RoboDK station: paint_robot.rdk

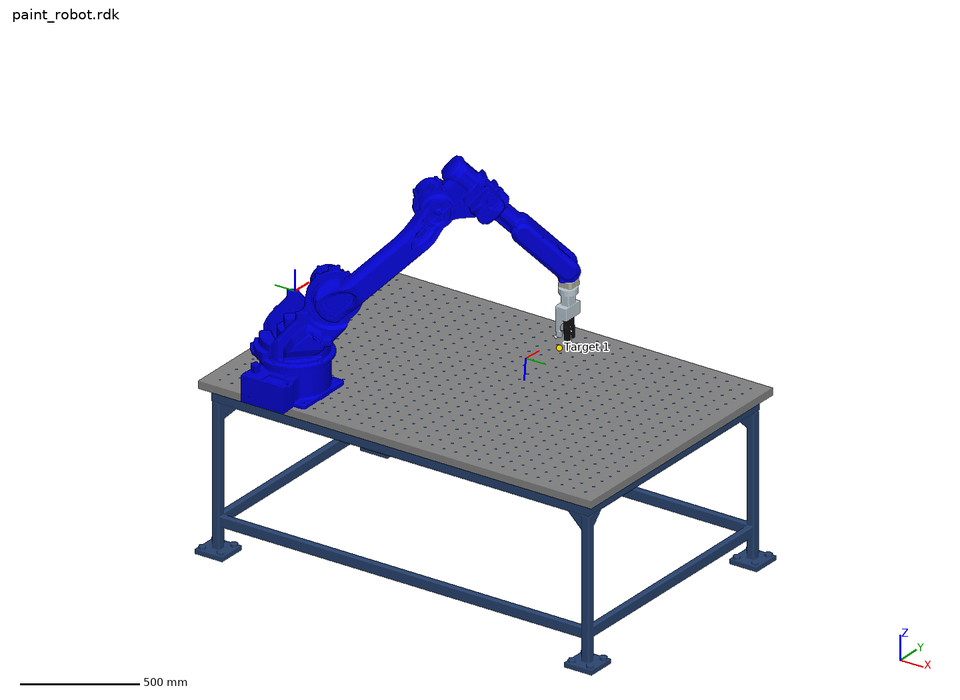
[picture v0: the station drawn from its stored meshes, robots at their saved joint values, targets as dots, program paths as lines]
Station paint_robot (saved by RoboDK 5.9.4). Poses are relative to the parent item; angles as X-Y-Z fixed-axis rotations.
  - frame Motoman HP6 Base at (2.87, -486.59, 450) mm, rotated rx 0 ry 0 rz 90.34 deg
    - robot Motoman HP6: 6 axes, payload 6 kg, reach 1378 mm, repeatability 0.08 mm, weight 130 kg
        modified DH rows (alpha deg, a mm, theta deg, d mm): 0, 0, 0, 450; -90, 150, -90, 0; 0, 570, 0, 0; -90, 155, 0, 640; 90, 0, 90, 0; -90, 0, 0, 95
        base shift (0, 0, -450) mm
        joint limits [-170, -90, -175, -180, -45, -360] to [170, 155, 250, 180, 225, 360]; home [0, 0, 0, 0, 0, 0]; saved at [-45.466, 50.692, 5.583, -1.431, 46.54, -134.308]
      - tool marker, TCP at (44.76, 5.33, 242.91) mm, size 100 x 89.2 x 281.5 mm
  - object table_draw at (0, 0, 0) mm, size 2020 x 1340 x 800 mm, geometry from Table-2000x1200x800mm.sld
  - frame Frame 2 at (685.28, 213.49, 50.15) mm, rotated rx -179.63 ry 3.79 rz 90.34 deg
    - target Target 1 (Cartesian target) at (108.07, 94.31, -36.38) mm, rotated rx 0.63 ry -5.51 rz -179.24 deg; joints [-43.036, 53.346, 5.286, -1.421, 49.532, -136.696] of Motoman HP6
  - Python program Prog1 (listed below)

--- Python program Prog1 ---
# draw_png_hp6_table_frame2.py
# Draw a PNG using Motoman HP6 in RoboDK (simulation).
# Station requirements:
#   Robot:       "Motoman HP6"
#   Tool:        "marker"
#   Draw frame:  "Frame 2"   -> XY plane of the paper
#   Base target: "DrawBase"  -> TCP at drawing height near center

from robolink import *   # RoboDK API
from robodk import *     # Pose tools
from robolink import TargetReachError

import cv2
import numpy as np
import os

# ---------------- CONFIG ----------------

IMAGE_PATH = r"vgtu.png"   # path to your PNG

ROBOT_NAME          = "Motoman HP6"
TOOL_NAME           = "marker"
DRAW_FRAME_NAME     = "Frame 2"
DRAW_BASE_TARGET    = "Target 1"

DRAW_AREA_MM = 150.0
MM_PER_PIXEL = 0.5     # scale of the drawing (mm per pixel)
POINT_STEP   = 4        # sample every Nth point of each contour

Z_DRAW  = 0.0           # drawing plane (relative to DrawBase)
Z_LIFT  = -50.0          # pen-up height above drawing plane (mm)

SPEED_DRAW   = 50.0     # mm/s when drawing
SPEED_TRAVEL = 200.0    # mm/s when travelling pen-up

# ----------------------------------------


def get_items(RDK: Robolink):
    """Get robot, tool, draw frame and base target from the station."""
    robot = RDK.Item(ROBOT_NAME, ITEM_TYPE_ROBOT)
    if not robot.Valid():
        raise Exception(f"Robot '{ROBOT_NAME}' not found in the station.")

    tool = RDK.Item(TOOL_NAME, ITEM_TYPE_TOOL)
    if not tool.Valid():
        raise Exception(f"Tool '{TOOL_NAME}' not found in the station.")

    draw_frame = RDK.Item(DRAW_FRAME_NAME, ITEM_TYPE_FRAME)
    if not draw_frame.Valid():
        raise Exception(f"Frame '{DRAW_FRAME_NAME}' (draw frame) not found.")

    base_target = RDK.Item(DRAW_BASE_TARGET, ITEM_TYPE_TARGET)
    if not base_target.Valid():
        raise Exception(
            f"Target '{DRAW_BASE_TARGET}' not found. "
            f"Teach it with the marker on the paper, near the center."
        )

    # Use our tool and draw frame for the robot
    robot.setPoseTool(tool)
    robot.setPoseFrame(draw_frame)

    return robot, draw_frame, base_target


def load_and_vectorize_image(image_path, draw_area_mm=DRAW_AREA_MM, point_step=4):
    """
    Load PNG, binarize it, find external contours and convert them
    to lists of XY points in mm, scaled to fit inside a square
    of size draw_area_mm x draw_area_mm and centered at (0,0).
    Returns: list of (N_i x 2) numpy arrays.
    """
    if not os.path.isfile(image_path):
        raise FileNotFoundError(f"Image not found: {image_path}")

    img = cv2.imread(image_path, cv2.IMREAD_GRAYSCALE)
    if img is None:
        raise Exception(f"Failed to read image: {image_path}")

    h, w = img.shape

    # Threshold: dark pixels become "ink"
    _, th = cv2.threshold(img, 200, 255, cv2.THRESH_BINARY_INV)

    contours, _ = cv2.findContours(th, cv2.RETR_EXTERNAL, cv2.CHAIN_APPROX_NONE)

    if not contours:
        raise Exception(
            "No drawing paths found in the image. "
            "Is the image mostly white/empty or too light?"
        )

    # --- collect all contour points in pixels to compute bounding box ---
    all_x = []
    all_y = []
    for cnt in contours:
        if len(cnt) < 5:
            continue
        xs = cnt[:, 0, 0]
        ys = cnt[:, 0, 1]
        all_x.append(xs)
        all_y.append(ys)

    all_x = np.concatenate(all_x).astype(np.float32)
    all_y = np.concatenate(all_y).astype(np.float32)

    xmin, xmax = all_x.min(), all_x.max()
    ymin, ymax = all_y.min(), all_y.max()

    cx = 0.5 * (xmin + xmax)
    cy = 0.5 * (ymin + ymax)

    span_x = xmax - xmin
    span_y = ymax - ymin
    span = max(span_x, span_y, 1e-6)   # avoid /0

    # scale so max dimension = draw_area_mm
    scale = float(draw_area_mm) / span

    paths_mm = []

    for cnt in contours:
        if len(cnt) < 5:
            continue

        pts = []
        for i in range(0, len(cnt), point_step):
            x_px = float(cnt[i][0][0])
            y_px = float(cnt[i][0][1])

            # center and scale; flip Y so "up" in image is +Y in frame
            x_mm = (x_px - cx) * scale
            y_mm = (y_px - cy) * scale

            pts.append([x_mm, y_mm])

        if len(pts) > 1:
            paths_mm.append(np.array(pts, dtype=float))

    if not paths_mm:
        raise Exception("Contours found, but no paths after processing.")

    # Optional: debug print to see range
    all_mm = np.vstack(paths_mm)
    print(
        f"[DEBUG] Drawing bounds in mm: "
        f"X [{all_mm[:,0].min():.1f}, {all_mm[:,0].max():.1f}], "
        f"Y [{all_mm[:,1].min():.1f}, {all_mm[:,1].max():.1f}]"
    )

    return paths_mm

# --------- motion helpers ---------

def move_pen_up(robot, base_pose, x_mm, y_mm, z_lift=Z_LIFT, speed=SPEED_TRAVEL):
    """Lift the pen to a safe height above (x,y) using a JOINT move."""
    pose_safe = base_pose * transl(float(x_mm), float(y_mm), float(z_lift))
    robot.setSpeed(speed)
    try:
        robot.MoveJ(pose_safe)
    except TargetReachError as e:
        print(f"[WARN] Pen-up unreachable at ({x_mm:.1f},{y_mm:.1f},{z_lift:.1f}): {e}")


def move_pen_down(robot, base_pose, x_mm, y_mm, z_draw=Z_DRAW, speed=SPEED_DRAW):
    """Move the pen down to drawing plane at (x,y) using a LINEAR move."""
    pose_draw = base_pose * transl(float(x_mm), float(y_mm), float(z_draw))
    robot.setSpeed(speed)
    try:
        robot.MoveL(pose_draw)
    except TargetReachError as e:
        print(f"[WARN] Pen-down unreachable at ({x_mm:.1f},{y_mm:.1f},{z_draw:.1f}): {e}")


def draw_paths(robot, base_pose, contours_mm,
               z_lift=Z_LIFT, z_draw=Z_DRAW,
               speed_draw=SPEED_DRAW, speed_travel=SPEED_TRAVEL):
    """Draw all contours, lifting the pen between them."""
    for pts_mm in contours_mm:
        if pts_mm.shape[0] < 2:
            continue

        # Start of contour
        x0, y0 = pts_mm[0]

        # Pen up → above first point
        move_pen_up(robot, base_pose, x0, y0, z_lift=z_lift, speed=speed_travel)

        # Pen down → drawing height
        move_pen_down(robot, base_pose, x0, y0, z_draw=z_draw, speed=speed_draw)

        # Follow contour
        for x_mm, y_mm in pts_mm[1:]:
            pose_target = base_pose * transl(float(x_mm), float(y_mm), float(z_draw))
            robot.setSpeed(speed_draw)
            try:
                robot.MoveL(pose_target)
            except TargetReachError:
                print(f"[WARN] Skipping unreachable point ({x_mm:.1f},{y_mm:.1f})")
                continue

        # Pen up at end of contour
        xe, ye = pts_mm[-1]
        move_pen_up(robot, base_pose, xe, ye, z_lift=z_lift, speed=speed_travel)


# --------------- main ----------------

def main():
    RDK = Robolink()

    robot, draw_frame, base_target = get_items(RDK)

    # Base pose gives us orientation and reference for (x,y,z) offsets
    base_pose = base_target.Pose()

    RDK.ShowMessage("Loading and vectorizing image...", False)
    contours_mm = load_and_vectorize_image(
    IMAGE_PATH,
    draw_area_mm=DRAW_AREA_MM,
    point_step=POINT_STEP,
    )

    RDK.ShowMessage(f"Found {len(contours_mm)} contours. Starting drawing...", False)

    draw_paths(
        robot,
        base_pose,
        contours_mm,
        z_lift=Z_LIFT,
        z_draw=Z_DRAW,
        speed_draw=SPEED_DRAW,
        speed_travel=SPEED_TRAVEL,
    )

    RDK.ShowMessage("Drawing complete (simulation).", False)


if __name__ == "__main__":
    main()
